// TIA Portal V17 export
// export: Created 2025-03-07T09:24:32.0698134Z, ExportSetting WithDefaults, DisplayName Totally Integrated Automation Portal, DisplayVersion V17 Update 8, DisplayName TIA Portal Openness, DisplayVersion V17 Update 8, DisplayName TIA Portal Version Control Interface, DisplayVersion V17, DisplayName SINAMICS Startdrive Advanced, DisplayVersion V17 SP2, DisplayName SINAMICS Startdrive G110M, G120, G120C, G120D, G120P, G115D, DisplayVersion V17 SP2, DisplayName SINAMICS Startdrive G130, G150, S120, S150, SINAMICS MV, S210, DisplayVersion V17 SP2, DisplayName STEP 7 Professional, DisplayVersion V17 Update 8, DisplayName SINUMERIK ONE STEP 7 Toolbox, DisplayVersion V17 Update 12, DisplayName SINUMERIK 840D sl STEP 7 Toolbox, DisplayVersion V17 Update 12, DisplayName STEP 7 Safety, DisplayVersion V17 Update 6, DisplayName WinCC Advanced, DisplayVersion V17 Update 8
VAR_GLOBAL   // PLC tag table "TAGS_IO_POWDER_FEEDERS_CLADDING"
   "//////////PF_HOPPERS_PRESSURE_SENSORS//////////" AT %M810.0 : Bool;
   "//////////POWDER_FEEDER_WEIGHT_CONTROL//////////" AT %M712.0 : Bool;
   "//////////POWDER_FLOW_SENSORS//////////" AT %M700.0 : Bool;
   U01_PF_1_WEIGHT_SENSOR_I AT %IW712 : Word;   // UNIT 01 POWDER FEEDER 1 WEIGHT SENSOR INPUT
   U02_COMBINER_FLOW_SENSOR_I AT %IW1706 : Word;   // UNIT 02 COMBINER FLOW SENSOR INPUT
   U02_OERLIKON_2_LINE_2_MEDICOAT_FLOW_CONTROL AT %MW16 : UInt;   // UNIT 02 OERLIKON 2 LINE 2 MEDICOAT FLOW CONTROL
   U02_OERLIKON_1_LINE_1_MEDICOAT_FLOW_CONTROL AT %IW1700 : Int;   // UNIT 02 OERLIKON 1 LINE 1 MEDICOAT FLOW CONTROL
   U02_COMBINER_MEDICOAT_FLOW_CONTROL AT %IW1708 : Int;   // UNIT 02 COMBINER MEDICOAT FLOW CONTROL
   U02_OERLIKON_2_LINE_1_MEDICOAT_FLOW_CONTROL AT %IW1704 : Int;   // UNIT 02 OERLIKON 2 LINE 1 MEDICOAT FLOW CONTROL
   U01_OERLIKON_1_LINE_1_MEDICOAT_FLOW_CONTROL AT %IW700 : Int;   // UNIT 01 OERLIKON 1 LINE 1 MEDICOAT FLOW CONTROL
   U02_PF_1_HPPR_1_PRESSURE_SENSOR_I AT %IW1818 : Word;   // UNIT 02 POWDER FEEDER 1 HOPPER 1 PRESSURE SENSOR INPUT
   U01_PF_1_HPPR_1_FLOW_SENSOR_I AT %MW700 : Word;   // UNIT 01 POWDER FEEDER 1 HOPPER 1 FLOW SENSOR INPUT
   U02_PF_2_HPPR_1_FLOW_SENSOR_I AT %MW1704 : Word;   // UNIT 02 POWDER FEEDER 2 HOPPER 1 FLOW SENSOR INPUT
   U01_PF_1_HPPR_1_PRESSURE_SENSOR_I AT %IW810 : Word;   // UNIT 01 POWDER FEEDER 1 HOPPER 1 PRESSURE SENSOR INPUT
   U02_PF_1_WEIGHT_SENSOR_I AT %MW1712 : Word;   // UNIT 02 POWDER FEEDER 1 WEIGHT SENSOR INPUT
   U02_PF_2_HPPR_1_PRESSURE_SENSOR_I AT %IW1822 : Word;   // UNIT 02 POWDER FEEDER 2 HOPPER 1 PRESSURE SENSOR INPUT
   U02_LASER_HEAD_FLOW_SENSOR_I AT %MW1708 : Word;   // UNIT 02 LASER HEAD FLOW SENSOR INPUT
   U02_PF_1_HPPR_2_PRESSURE_SENSOR_I AT %IW1820 : Word;   // UNIT 02 POWDER FEEDER 1 HOPPER 2 PRESSURE SENSOR INPUT
   U01_PF_1_HPPR_2_PRESSURE_SENSOR_I AT %IW812 : Word;   // UNIT 01 POWDER FEEDER 1 HOPPER 2 PRESSURE SENSOR INPUT
   U02_OERLIKON_1_LINE_2_MEDICOAT_FLOW_CONTROL AT %IW1702 : Int;   // UNIT 02 OERLIKON 1 LINE 2 MEDICOAT FLOW CONTROL
   U01_LASER_HEAD_FLOW_SENSOR_I AT %MW706 : Word;   // UNIT 01 LASER HEAD FLOW SENSOR INPUT
   U02_PF_2_WEIGHT_SENSOR_I AT %MW1714 : Word;   // UNIT 02 POWDER FEEDER 2 WEIGHT SENSOR INPUT
   U01_COMBINER_MEDICOAT_FLOW_CONTROL AT %IW708 : Int;   // UNIT 01 COMBINER MEDICOAT FLOW CONTROL
   U02_LASER_HEAD_MEDICOAT_CONTROL AT %IW1710 : Int;   // UNIT 02 LASER HEAD MEDICOAT FLOW CONTROL
   U01_COMBINER_FLOW_SENSOR_I AT %MW704 : Word;   // UNIT 01 COMBINER FLOW SENSOR INPUT
   U02_PF_1_HPPR_2_FLOW_SENSOR_I AT %MW1702 : Word;   // UNIT 02 POWDER FEEDER 1 HOPPER 2 FLOW SENSOR INPUT
   U01_OERLIKON_1_LINE_2_MEDICOAT_FLOW_CONTROL AT %IW702 : Int;   // UNIT 01 OERLIKON 1 LINE 2 MEDICOAT FLOW CONTROL
   U01_PF_1_HPPR_2_FLOW_SENSOR_I AT %MW702 : Word;   // UNIT 01 POWDER FEEDER 1 HOPPER 2 FLOW SENSOR INPUT
   U02_PF_1_HPPR_1_FLOW_SENSOR_I AT %MW1700 : Word;   // UNIT 02 POWDER FEEDER 1 HOPPER 1 FLOW SENSOR INPUT
   U01_LASER_HEAD_MEDICOAT_CONTROL AT %IW710 : Int;   // UNIT 01 LASER HEAD MEDICOAT FLOW CONTROL
   U02_PF1_L2_STIRRER_CURRENT AT %IW1716 : Int;
   U02_PF1_L1_STIRRER_CURRENT AT %IW1712 : Int;
   U02_PF2_L1_DISK_CURRENT AT %IW1722 : Int;
   U02_PF2_L1_STIRRER_CURRENT AT %IW1720 : Int;
   U02_PF1_L2_DISK_CURRENT AT %IW1718 : Int;
   U01_PF1_L2_DISK_CURRENT AT %IW722 : Int;
   U01_PF1_L1_DISK_CURRENT AT %IW718 : Int;
   U01_PF1_L2_STIRRER_CURRENT AT %IW720 : Int;
   U01_PF1_L1_STIRRER_CURRENT AT %IW716 : Int;
   U02_PF1_L1_DISK_CURRENT AT %IW1714 : Int;
END_VAR
